{attribute 'qualified_only'}
{attribute 'strict'}
TYPE E_Message_Generator :
(
	eNoMessage := 0,
	eTooMuchGenerators := 1,
	eGeneratorError := 2,
	eNoConnectionToBackend := 3
);
END_TYPE

(* stored: Version 1.1.0.1, ProductVersion 3.1.4024.6
   DUT E_Message_Generator: Id {45cefac7-7d01-4681-8272-8200b9ec6ebb} *)
